Yaskawa INFORM job: R1_W66-W67(-70,-90)KM-OK.JBI

/JOB
//NAME R1_W66-W67(-70,-90)KM-OK
///FOLDERNAME KRIS-SCIANA
//POS
///NPOS 41,41,0,3,0,0
///TOOL 0
///POSTYPE PULSE
///PULSE
C00000=135635,-24500,-41716,-31750,82638,-33791
C00001=121173,28136,37388,-9783,95382,-11090
C00002=121152,31888,45574,-9734,92313,-10856
C00003=121142,35145,50794,-9721,90794,-10743
C00004=121143,35483,52754,-9718,89774,-10663
C00005=121143,35225,52204,-9718,89977,-10679
C00006=121140,38719,56440,-9718,89178,-10618
C00007=121176,37573,54181,-9710,89973,-10668
C00008=120187,34889,50757,-9920,90573,-11044
C00009=119360,34923,50783,-10093,90475,-11313
C00010=120187,34889,50757,-9920,90573,-11044
C00011=120195,33129,47147,-9931,91873,-11144
C00012=120213,29283,38831,-9979,94971,-11386
C00013=124262,41791,46564,15679,81195,-12986
C00014=125301,47706,56682,15822,77923,-13043
C00015=124319,51586,62900,15917,76347,-13598
C00016=124340,50707,62802,15941,75964,-13642
C00017=124340,50450,62252,15928,76164,-13616
C00018=124303,54143,66935,15991,75223,-13754
C00019=124340,48208,57292,15821,77994,-13376
C00020=118829,36803,52428,28844,69518,-21730
C00021=119649,36749,52382,28805,69244,-21478
C00022=118829,36803,52428,28844,69518,-21730
C00023=118147,34363,48669,28702,70681,-21695
C00024=116410,28824,40027,28425,73448,-21667
C00025=120722,36277,52307,-21922,60833,8108
C00026=120727,-61195,-31383,-21647,62154,7841
C00027=109986,44671,45472,-4739,72285,-39309
C00028=109829,25936,29329,-1019,58563,-75027
C00029=109983,-48218,-17757,-10134,60962,2786
C00030=106347,-42262,-11385,-6074,61232,1020
C00031=120730,33890,48639,-21720,61795,7914
C00032=120725,33272,48739,-21793,61440,7984
C00033=75989,-14815,16193,34885,81654,-11665
C00034=122712,-37532,556,36823,59959,421
C00035=127515,-37153,788,36460,58070,1866
C00036=130523,-28224,-7066,20648,68494,-3594
C00037=128165,9668,-249,4290,62701,-67347
C00038=132020,10447,-13346,2437,70990,-65718
C00039=130510,-84668,-101602,2499,71155,-65752
C00040=130510,-84668,-101602,2499,71155,-65752
BC00000=108350,470429,937615
BC00001=156279,382090,733616
BC00002=156279,382090,733616
BC00003=156279,382090,733616
BC00004=156279,382090,733616
BC00005=156279,382090,733616
BC00006=156279,382090,733616
BC00007=156279,382090,733616
BC00008=156279,382090,733616
BC00009=156279,382090,733616
BC00010=156279,382090,733616
BC00011=156279,382090,733616
BC00012=156279,382090,733616
BC00013=113113,427324,688648
BC00014=113113,427324,688648
BC00015=113113,427324,688648
BC00016=113113,427324,688648
BC00017=113113,427324,688648
BC00018=113113,427324,688648
BC00019=113113,427324,688648
BC00020=113113,427324,688648
BC00021=113113,427324,688648
BC00022=113113,427324,688648
BC00023=113113,427324,688648
BC00024=113113,427324,688648
BC00025=131179,446202,829365
BC00026=131601,347931,721839
BC00027=135449,439844,694419
BC00028=135449,439844,694419
BC00029=131601,347931,721839
BC00030=131601,347931,721839
BC00031=135449,439844,694419
BC00032=135449,439844,694419
BC00033=131601,347931,721839
BC00034=131602,347960,721830
BC00035=131602,347960,721830
BC00036=132199,362211,717578
BC00037=135448,439845,694416
BC00038=135448,439845,694416
BC00039=135448,439845,876221
BC00040=135448,596711,876221
///POSTYPE BASE
///RECTAN
///RCONF 0,0,0,0,1,0,0,0,0,0,0,0,0,0,0,0,0,0,0,0,0,0,0,0
P00006=2.006,1.622,-0.565,0.0000,0.0000,0.0000
P00021=0.073,2.058,-0.109,0.0000,0.0000,0.0000
P00022=2.006,1.622,-0.565,0.0000,0.0000,0.0000
//INST
///DATE 2025/04/14 13:30
///ATTR SC,RW
///GROUP1 RB1,BS1
NOP
'r2_W66-W67(-70,-90)
MOVJ C00000 BC00000 VJ=50.00
'Path S1112 (for W504)
SFTOF
MOVJ C00001 BC00001 VJ=80.00
MOVJ C00002 BC00002 VJ=100.00
MOVL C00003 BC00003 V=60.0
REFP 3 C00004 BC00004
CALL JOB:SEARCH-R1
SET P021 P006
SFTON P021
MOVL C00005 BC00005 V=60.0
REFP 3 C00006 BC00006
CALL JOB:SEARCH-R1
SET P021 P006
SFTON P021
MOVL C00007 BC00007 V=60.0
MOVL C00008 BC00008 V=60.0
REFP 3 C00009 BC00009
CALL JOB:SEARCH-R1
SET P021 P006
SFTON P021
MOVL C00010 BC00010 V=60.0
MOVL C00011 BC00011 V=100.0
MOVL C00012 BC00012 V=100.0
'Path S1113 (for W504)
SFTOF
MOVJ C00013 BC00013 VJ=100.00
MOVJ C00014 BC00014 VJ=100.00
MOVL C00015 BC00015 V=60.0
REFP 3 C00016 BC00016
CALL JOB:SEARCH-R1
SET P022 P006
SFTON P022
MOVL C00017 BC00017 V=60.0
REFP 3 C00018 BC00018
CALL JOB:SEARCH-R1
SET P022 P006
SFTON P022
MOVL C00019 BC00019 V=60.0
MOVL C00020 BC00020 V=60.0
REFP 3 C00021 BC00021
CALL JOB:SEARCH-R1
SET P022 P006
SFTON P022
MOVL C00022 BC00022 V=60.0
MOVL C00023 BC00023 V=100.0
MOVL C00024 BC00024 V=100.0
'Path W1114
SFTOF
SFTON P021
CALL JOB:COFNIJ_DRUT
MOVJ C00025 BC00025 VJ=100.00
MOVJ C00026 BC00026 VJ=100.00
COMM MOVJ C00027 BC00027 VJ=100.00
COMM MOVJ C00028 BC00028 VJ=100.00
MOVL C00029 BC00029 V=333.3
MOVL C00030 BC00030 V=100.0 PL=0
REFP 1 C00031 BC00031
REFP 2 C00032 BC00032
MACRO1 MJ#(0) ARGF7
ARCON
MOVL C00033 BC00033 V=11.2
SFTON P022
MOVL C00034 BC00034 V=10.8
MOVL C00035 BC00035 V=10.8
ARCOF
MOVL C00036 BC00036 V=100.0
SFTOF
MOVL C00037 BC00037 V=100.0
MOVJ C00038 BC00038 VJ=100.00
MOVJ C00039 BC00039 VJ=100.00
MOVJ C00040 BC00040 VJ=100.00
END
